// TIA Portal V20 export
// export: Created 2026-07-16T23:20:27.074812Z, ExportSetting WithDefaults, DisplayName Totally Integrated Automation Portal, DisplayVersion V20 Update 5, DisplayName TIA Portal Openness, DisplayVersion V20 Update 4, DisplayName TIA Portal Version Control Interface, DisplayVersion V20 Update 5, DisplayName SINAMICS Startdrive Advanced, DisplayVersion V20, DisplayName SINAMICS DCC, DisplayVersion V20, DisplayName SINAMICS Startdrive G130, G150, S120, S150, SINAMICS MV, G220, S200, S210, DisplayVersion V20, DisplayName SINAMICS Startdrive G110M, G120, G120C, G120D, G120P, G115D, DisplayVersion V20, DisplayName STEP 7 Professional, DisplayVersion V20 Update 5, DisplayName STEP 7 Safety, DisplayVersion V20 Update 2, DisplayName WinCC Basic/Comfort/Advanced, DisplayVersion V20 Update 5, DisplayName WinCC Unified, DisplayVersion V20 Update 5
DATA_BLOCK "iDB_MotorFwdRevSystem_Shredder"   // DB6
VERSION : 0.1
// stored: AutoNumber true, DBAccessibleFromOPCUA true, InstanceOfName FB_MotorFwdRevSystem, InstanceOfType FB
"FB_MotorFwdRevSystem"
   // VAR RETAIN
   //    IO : "MotorFwdRevIOSet";
   // END_VAR
   // VAR
   //    RisingEdgeFlags : Array[0..3] of Bool;
   //    NegitiveSignalEdge : Array[0..2] of Bool;
   //    Pasue : Bool;
   //    HrTotaliserTimerReset : Bool;
   //    EnableUPSTimeMS : DInt;
   //    ShutdownTimeMS : DInt;
   //    FTTimeMS : DInt;
   //    PauseTimeMS : DInt;
   //    ReverseIgnoreFTTimeMS : DInt;
   //    FaultTripTimer { S7_SetPoint := 'True'} : TON_TIME;
   //    FTSTimer { S7_SetPoint := 'True'} : TON_TIME;
   //    EnableUpstreamTimer { S7_SetPoint := 'True'} : TON_TIME;
   //    ShutdownTimer { S7_SetPoint := 'True'} : TON_TIME;
   //    GeneralDelayTimer { S7_SetPoint := 'True'} : TON_TIME;
   //    InHandReqPreStart { S7_SetPoint := 'True'} : TON_TIME;
   //    CycleDelayReset { S7_SetPoint := 'True'} : TON_TIME;
   // END_VAR
   // VAR RETAIN
   //    HrTotaliserTimer { S7_SetPoint := 'True'} : TONR_TIME;
   // END_VAR
   // VAR
   //    ReversalPauseTimer { S7_SetPoint := 'True'} : TON_TIME;
   //    ReversalIgnoreFTTimer { S7_SetPoint := 'True'} : TON_TIME;
   //    PreStartMemory { S7_SetPoint := 'True'} : Bool;
   //    HandPosEdge : Bool;
   //    HandNegEdge : Bool;
   //    CycleDelay : Bool;
   // END_VAR
BEGIN
   IO.FTTime := 10.0;
   IO.ReverseDelay := 8.0;
   IO.ReverseIgnoreFT := 12.0;
END_DATA_BLOCK
